// TIA Portal V15.1 export
// export: Created 2024-05-17T05:38:59.7002443Z, ExportSetting WithDefaults, DisplayName Totally Integrated Automation Portal, DisplayVersion V15.1 Update 5, DisplayName TIA Portal Openness, DisplayVersion V15.1 Update 5, DisplayName SINAMICS Startdrive Advanced, DisplayVersion V15.1, DisplayName G130, G150, S120, S150, SINAMICS MV, S210, DisplayVersion V15.1, DisplayName G110M, G120, G120C, G120D, G120P, DisplayVersion V15.1, DisplayName STEP 7 Professional, DisplayVersion V15.1 Update 5, DisplayName STEP 7 Safety, DisplayVersion V15.1, DisplayName WinCC Professional, DisplayVersion V15.1 Update 5, DisplayName SIMATIC Visualization Architect, DisplayVersion V15.1
FUNCTION "209000NCP01ComVD" : Void   // FC256, FBD
TITLE = 209000NCP01ComSafety
{ S7_Optimized_Access := 'FALSE' }
AUTHOR : VCC
VERSION : 0.1
// stored: AutoNumber false, IsIECCheckEnabled false, SetENOAutomatically False, UDAEnableTagReadback false
   VAR_OUTPUT
      O_AlarmA : Bool;   // Alarm A
      O_AlarmB : Bool;   // Alarm B
      O_AlarmC : Bool;   // Alarm C
      O_AlarmD : Bool;   // Alarm D
      O_AlarmABCondition : Bool;   // Alarm AB Condition
      H_IAnim : Word;   // Icon Animation
   END_VAR
BEGIN

REGION Network 1: **** 1 - Inputs **** VD Config Alarm Reporting
   // Communication With VD Alarm Instance
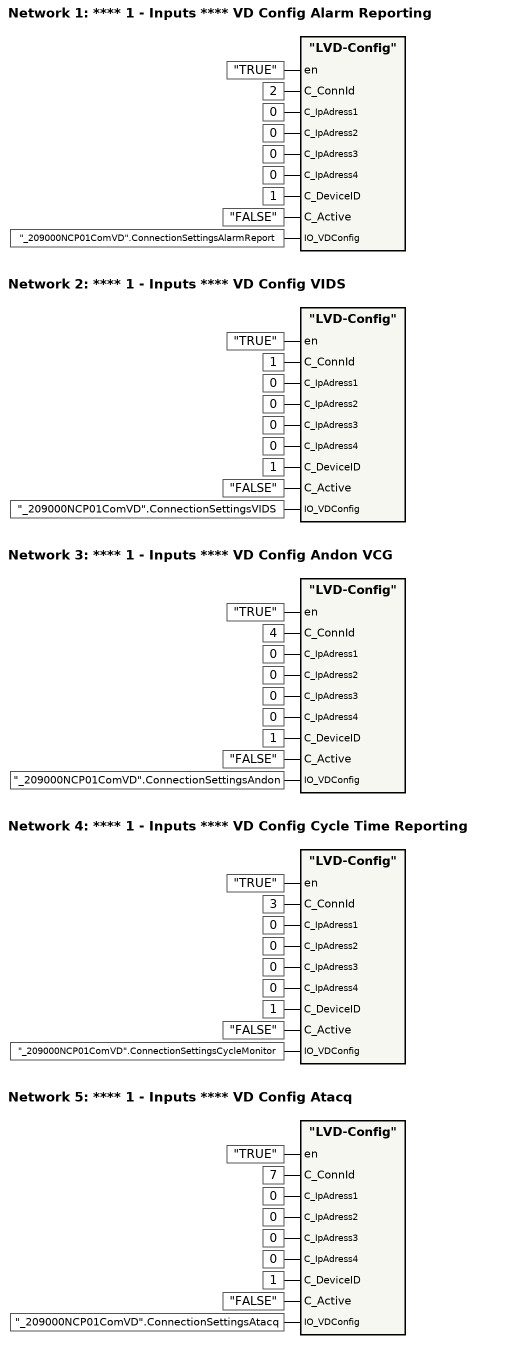
   IF "TRUE" THEN
       "LVD-Config"(C_ConnId := 2,
                    C_IpAdress1 := 0,
                    C_IpAdress2 := 0,
                    C_IpAdress3 := 0,
                    C_IpAdress4 := 0,
                    C_DeviceID := 1,
                    C_Active := "FALSE",
                    IO_VDConfig := "_209000NCP01ComVD".ConnectionSettingsAlarmReport);
   END_IF;
END_REGION

REGION Network 2: **** 1 - Inputs **** VD Config VIDS
   // Communication with VD Prod Instance
   IF "TRUE" THEN
       "LVD-Config"(C_ConnId := 1,
                    C_IpAdress1 := 0,
                    C_IpAdress2 := 0,
                    C_IpAdress3 := 0,
                    C_IpAdress4 := 0,
                    C_DeviceID := 1,
                    C_Active := "FALSE",
                    IO_VDConfig := "_209000NCP01ComVD".ConnectionSettingsVIDS);
   END_IF;
END_REGION

REGION Network 3: **** 1 - Inputs **** VD Config Andon VCG
   // Communication with VD Andon Instance
   IF "TRUE" THEN
       "LVD-Config"(C_ConnId := 4,
                    C_IpAdress1 := 0,
                    C_IpAdress2 := 0,
                    C_IpAdress3 := 0,
                    C_IpAdress4 := 0,
                    C_DeviceID := 1,
                    C_Active := "FALSE",
                    IO_VDConfig := "_209000NCP01ComVD".ConnectionSettingsAndon);
   END_IF;
END_REGION

REGION Network 4: **** 1 - Inputs **** VD Config Cycle Time Reporting
   // Communication setup for cycle time reporting
   IF "TRUE" THEN
       "LVD-Config"(C_ConnId := 3,
                    C_IpAdress1 := 0,
                    C_IpAdress2 := 0,
                    C_IpAdress3 := 0,
                    C_IpAdress4 := 0,
                    C_DeviceID := 1,
                    C_Active := "FALSE",
                    IO_VDConfig := "_209000NCP01ComVD".ConnectionSettingsCycleMonitor);
   END_IF;
END_REGION

REGION Network 5: **** 1 - Inputs **** VD Config Atacq
   // Communication setup for Atacq reporting
   IF "TRUE" THEN
       "LVD-Config"(C_ConnId := 7,
                    C_IpAdress1 := 0,
                    C_IpAdress2 := 0,
                    C_IpAdress3 := 0,
                    C_IpAdress4 := 0,
                    C_DeviceID := 1,
                    C_Active := "FALSE",
                    IO_VDConfig := "_209000NCP01ComVD".ConnectionSettingsAtacq);
   END_IF;
END_REGION

REGION Network 6: **** 1 - Inputs **** VD Config Logistic
   // Communication setup for Logistic reporting
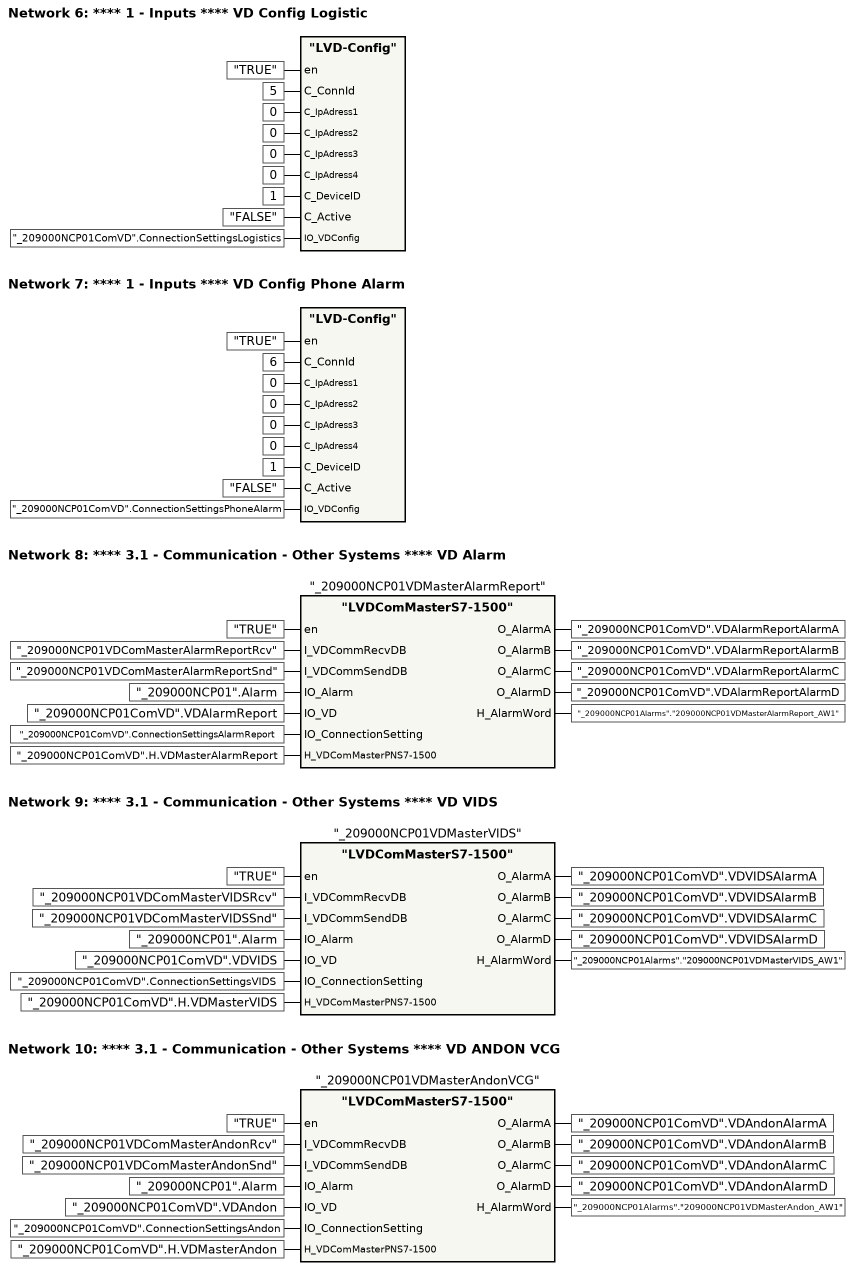
   IF "TRUE" THEN
       "LVD-Config"(C_ConnId := 5,
                    C_IpAdress1 := 0,
                    C_IpAdress2 := 0,
                    C_IpAdress3 := 0,
                    C_IpAdress4 := 0,
                    C_DeviceID := 1,
                    C_Active := "FALSE",
                    IO_VDConfig := "_209000NCP01ComVD".ConnectionSettingsLogistics);
   END_IF;
END_REGION

REGION Network 7: **** 1 - Inputs **** VD Config Phone Alarm
   // Communication setup for Phone Alarm
   IF "TRUE" THEN
       "LVD-Config"(C_ConnId := 6,
                    C_IpAdress1 := 0,
                    C_IpAdress2 := 0,
                    C_IpAdress3 := 0,
                    C_IpAdress4 := 0,
                    C_DeviceID := 1,
                    C_Active := "FALSE",
                    IO_VDConfig := "_209000NCP01ComVD".ConnectionSettingsPhoneAlarm);
   END_IF;
END_REGION

REGION Network 8: **** 3.1 - Communication - Other Systems **** VD Alarm
   // Connection VD Alarm
   IF "TRUE" THEN
       "_209000NCP01VDMasterAlarmReport"(I_VDCommRecvDB := "_209000NCP01VDComMasterAlarmReportRcv",   // "LVDComMasterS7-1500"
                               I_VDCommSendDB := "_209000NCP01VDComMasterAlarmReportSnd",
                               IO_Alarm := "_209000NCP01".Alarm,
                               IO_VD := "_209000NCP01ComVD".VDAlarmReport,
                               IO_ConnectionSetting := "_209000NCP01ComVD".ConnectionSettingsAlarmReport,
                               "H_VDComMasterPNS7-1500" := "_209000NCP01ComVD".H.VDMasterAlarmReport,
                               O_AlarmA => "_209000NCP01ComVD".VDAlarmReportAlarmA,
                               O_AlarmB => "_209000NCP01ComVD".VDAlarmReportAlarmB,
                               O_AlarmC => "_209000NCP01ComVD".VDAlarmReportAlarmC,
                               O_AlarmD => "_209000NCP01ComVD".VDAlarmReportAlarmD,
                               H_AlarmWord => "_209000NCP01Alarms"."209000NCP01VDMasterAlarmReport_AW1");
   END_IF;
END_REGION

REGION Network 9: **** 3.1 - Communication - Other Systems **** VD VIDS
   // Connection VD Production System
   IF "TRUE" THEN
       "_209000NCP01VDMasterVIDS"(I_VDCommRecvDB := "_209000NCP01VDComMasterVIDSRcv",   // "LVDComMasterS7-1500"
                               I_VDCommSendDB := "_209000NCP01VDComMasterVIDSSnd",
                               IO_Alarm := "_209000NCP01".Alarm,
                               IO_VD := "_209000NCP01ComVD".VDVIDS,
                               IO_ConnectionSetting := "_209000NCP01ComVD".ConnectionSettingsVIDS,
                               "H_VDComMasterPNS7-1500" := "_209000NCP01ComVD".H.VDMasterVIDS,
                               O_AlarmA => "_209000NCP01ComVD".VDVIDSAlarmA,
                               O_AlarmB => "_209000NCP01ComVD".VDVIDSAlarmB,
                               O_AlarmC => "_209000NCP01ComVD".VDVIDSAlarmC,
                               O_AlarmD => "_209000NCP01ComVD".VDVIDSAlarmD,
                               H_AlarmWord => "_209000NCP01Alarms"."209000NCP01VDMasterVIDS_AW1");
   END_IF;
END_REGION

REGION Network 10: **** 3.1 - Communication - Other Systems **** VD ANDON VCG
   // Connection VD Andon System
   IF "TRUE" THEN
       "_209000NCP01VDMasterAndonVCG"(I_VDCommRecvDB := "_209000NCP01VDComMasterAndonRcv",   // "LVDComMasterS7-1500"
                               I_VDCommSendDB := "_209000NCP01VDComMasterAndonSnd",
                               IO_Alarm := "_209000NCP01".Alarm,
                               IO_VD := "_209000NCP01ComVD".VDAndon,
                               IO_ConnectionSetting := "_209000NCP01ComVD".ConnectionSettingsAndon,
                               "H_VDComMasterPNS7-1500" := "_209000NCP01ComVD".H.VDMasterAndon,
                               O_AlarmA => "_209000NCP01ComVD".VDAndonAlarmA,
                               O_AlarmB => "_209000NCP01ComVD".VDAndonAlarmB,
                               O_AlarmC => "_209000NCP01ComVD".VDAndonAlarmC,
                               O_AlarmD => "_209000NCP01ComVD".VDAndonAlarmD,
                               H_AlarmWord => "_209000NCP01Alarms"."209000NCP01VDMasterAndon_AW1");
   END_IF;
END_REGION

REGION Network 11: **** 3.1 - Communication - Other Systems **** VD Cycle Time Monitoring
   // Connection VD Cycle Time Monitoring
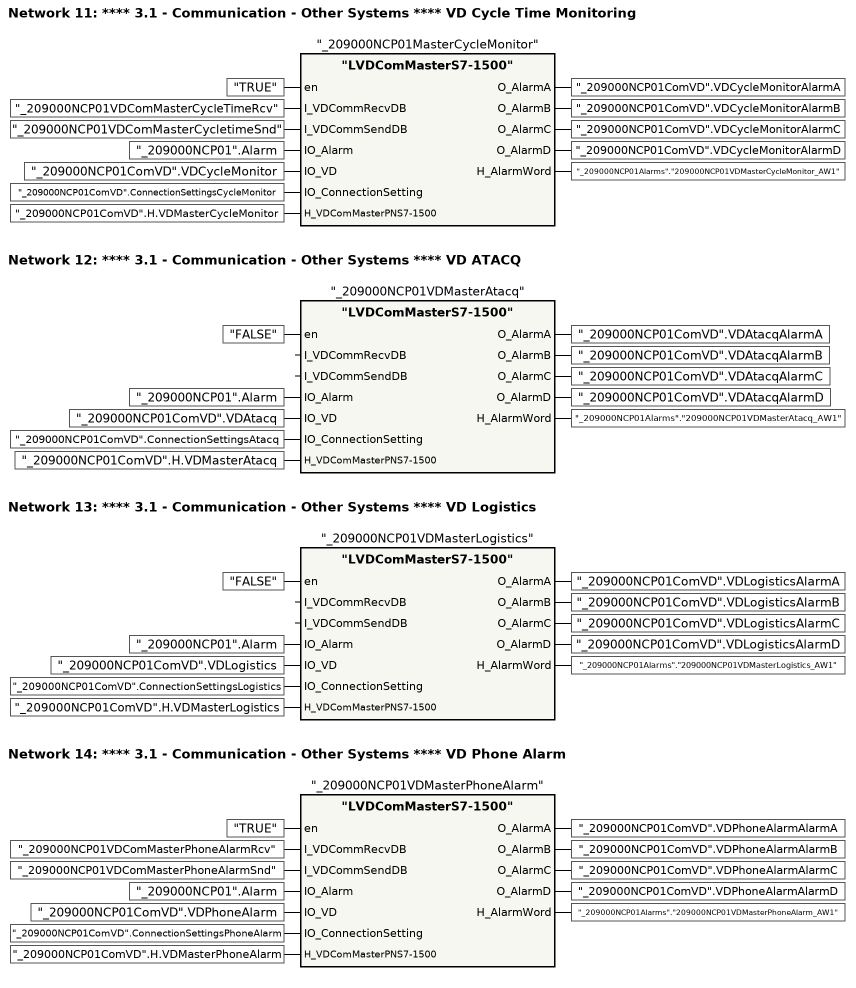
   IF "TRUE" THEN
       "_209000NCP01MasterCycleMonitor"(I_VDCommRecvDB := "_209000NCP01VDComMasterCycleTimeRcv",   // "LVDComMasterS7-1500"
                               I_VDCommSendDB := "_209000NCP01VDComMasterCycletimeSnd",
                               IO_Alarm := "_209000NCP01".Alarm,
                               IO_VD := "_209000NCP01ComVD".VDCycleMonitor,
                               IO_ConnectionSetting := "_209000NCP01ComVD".ConnectionSettingsCycleMonitor,
                               "H_VDComMasterPNS7-1500" := "_209000NCP01ComVD".H.VDMasterCycleMonitor,
                               O_AlarmA => "_209000NCP01ComVD".VDCycleMonitorAlarmA,
                               O_AlarmB => "_209000NCP01ComVD".VDCycleMonitorAlarmB,
                               O_AlarmC => "_209000NCP01ComVD".VDCycleMonitorAlarmC,
                               O_AlarmD => "_209000NCP01ComVD".VDCycleMonitorAlarmD,
                               H_AlarmWord => "_209000NCP01Alarms"."209000NCP01VDMasterCycleMonitor_AW1");
   END_IF;
END_REGION

REGION Network 12: **** 3.1 - Communication - Other Systems **** VD ATACQ
   // Connection VD ATACQ
   IF "FALSE" THEN
       "_209000NCP01VDMasterAtacq"(IO_Alarm := "_209000NCP01".Alarm,   // "LVDComMasterS7-1500"
                               IO_VD := "_209000NCP01ComVD".VDAtacq,
                               IO_ConnectionSetting := "_209000NCP01ComVD".ConnectionSettingsAtacq,
                               "H_VDComMasterPNS7-1500" := "_209000NCP01ComVD".H.VDMasterAtacq,
                               O_AlarmA => "_209000NCP01ComVD".VDAtacqAlarmA,
                               O_AlarmB => "_209000NCP01ComVD".VDAtacqAlarmB,
                               O_AlarmC => "_209000NCP01ComVD".VDAtacqAlarmC,
                               O_AlarmD => "_209000NCP01ComVD".VDAtacqAlarmD,
                               H_AlarmWord => "_209000NCP01Alarms"."209000NCP01VDMasterAtacq_AW1");
   END_IF;
END_REGION

REGION Network 13: **** 3.1 - Communication - Other Systems **** VD Logistics
   // Connection VD Logistics
   IF "FALSE" THEN
       "_209000NCP01VDMasterLogistics"(IO_Alarm := "_209000NCP01".Alarm,   // "LVDComMasterS7-1500"
                               IO_VD := "_209000NCP01ComVD".VDLogistics,
                               IO_ConnectionSetting := "_209000NCP01ComVD".ConnectionSettingsLogistics,
                               "H_VDComMasterPNS7-1500" := "_209000NCP01ComVD".H.VDMasterLogistics,
                               O_AlarmA => "_209000NCP01ComVD".VDLogisticsAlarmA,
                               O_AlarmB => "_209000NCP01ComVD".VDLogisticsAlarmB,
                               O_AlarmC => "_209000NCP01ComVD".VDLogisticsAlarmC,
                               O_AlarmD => "_209000NCP01ComVD".VDLogisticsAlarmD,
                               H_AlarmWord => "_209000NCP01Alarms"."209000NCP01VDMasterLogistics_AW1");
   END_IF;
END_REGION

REGION Network 14: **** 3.1 - Communication - Other Systems **** VD Phone Alarm
   // Connection VD Phone Alarm
   IF "TRUE" THEN
       "_209000NCP01VDMasterPhoneAlarm"(I_VDCommRecvDB := "_209000NCP01VDComMasterPhoneAlarmRcv",   // "LVDComMasterS7-1500"
                               I_VDCommSendDB := "_209000NCP01VDComMasterPhoneAlarmSnd",
                               IO_Alarm := "_209000NCP01".Alarm,
                               IO_VD := "_209000NCP01ComVD".VDPhoneAlarm,
                               IO_ConnectionSetting := "_209000NCP01ComVD".ConnectionSettingsPhoneAlarm,
                               "H_VDComMasterPNS7-1500" := "_209000NCP01ComVD".H.VDMasterPhoneAlarm,
                               O_AlarmA => "_209000NCP01ComVD".VDPhoneAlarmAlarmA,
                               O_AlarmB => "_209000NCP01ComVD".VDPhoneAlarmAlarmB,
                               O_AlarmC => "_209000NCP01ComVD".VDPhoneAlarmAlarmC,
                               O_AlarmD => "_209000NCP01ComVD".VDPhoneAlarmAlarmD,
                               H_AlarmWord => "_209000NCP01Alarms"."209000NCP01VDMasterPhoneAlarm_AW1");
   END_IF;
END_REGION

REGION Network 15: **** 3.1 - Communication - Other Systems **** Phone Alarm Request
   // Phone alarm request
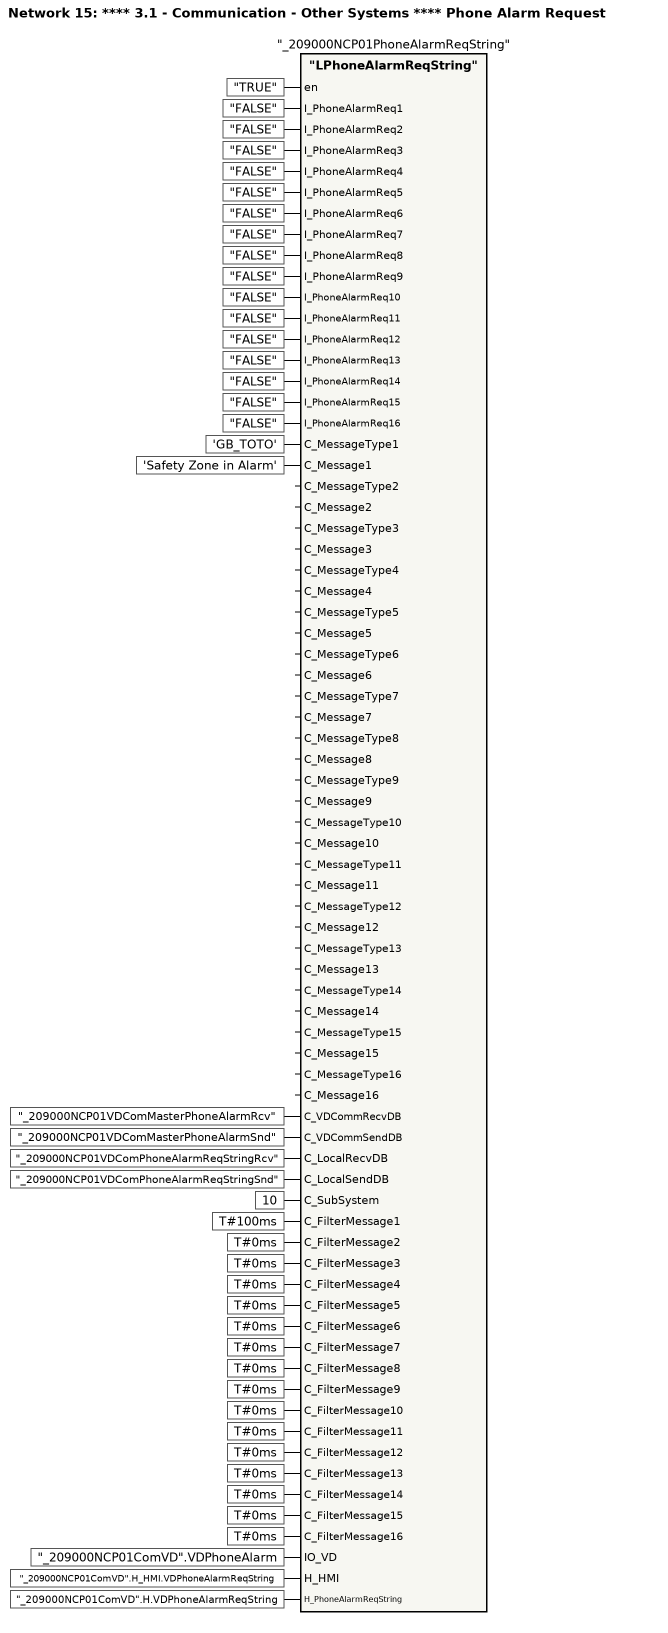
   IF "TRUE" THEN
       "_209000NCP01PhoneAlarmReqString"(I_PhoneAlarmReq1 := "FALSE",   // "LPhoneAlarmReqString"
                               I_PhoneAlarmReq2 := "FALSE",
                               I_PhoneAlarmReq3 := "FALSE",
                               I_PhoneAlarmReq4 := "FALSE",
                               I_PhoneAlarmReq5 := "FALSE",
                               I_PhoneAlarmReq6 := "FALSE",
                               I_PhoneAlarmReq7 := "FALSE",
                               I_PhoneAlarmReq8 := "FALSE",
                               I_PhoneAlarmReq9 := "FALSE",
                               I_PhoneAlarmReq10 := "FALSE",
                               I_PhoneAlarmReq11 := "FALSE",
                               I_PhoneAlarmReq12 := "FALSE",
                               I_PhoneAlarmReq13 := "FALSE",
                               I_PhoneAlarmReq14 := "FALSE",
                               I_PhoneAlarmReq15 := "FALSE",
                               I_PhoneAlarmReq16 := "FALSE",
                               C_MessageType1 := 'GB_TOTO',
                               C_Message1 := 'Safety Zone in Alarm',
                               C_VDCommRecvDB := "_209000NCP01VDComMasterPhoneAlarmRcv",
                               C_VDCommSendDB := "_209000NCP01VDComMasterPhoneAlarmSnd",
                               C_LocalRecvDB := "_209000NCP01VDComPhoneAlarmReqStringRcv",
                               C_LocalSendDB := "_209000NCP01VDComPhoneAlarmReqStringSnd",
                               C_SubSystem := 10,
                               C_FilterMessage1 := T#100ms,
                               C_FilterMessage2 := T#0ms,
                               C_FilterMessage3 := T#0ms,
                               C_FilterMessage4 := T#0ms,
                               C_FilterMessage5 := T#0ms,
                               C_FilterMessage6 := T#0ms,
                               C_FilterMessage7 := T#0ms,
                               C_FilterMessage8 := T#0ms,
                               C_FilterMessage9 := T#0ms,
                               C_FilterMessage10 := T#0ms,
                               C_FilterMessage11 := T#0ms,
                               C_FilterMessage12 := T#0ms,
                               C_FilterMessage13 := T#0ms,
                               C_FilterMessage14 := T#0ms,
                               C_FilterMessage15 := T#0ms,
                               C_FilterMessage16 := T#0ms,
                               IO_VD := "_209000NCP01ComVD".VDPhoneAlarm,
                               H_HMI := "_209000NCP01ComVD".H_HMI.VDPhoneAlarmReqString,
                               H_PhoneAlarmReqString := "_209000NCP01ComVD".H.VDPhoneAlarmReqString);
   END_IF;
END_REGION

REGION Network 16: **** 4.6 - Machine status - Indications **** Icon animation
   // Icon animation to WinCC
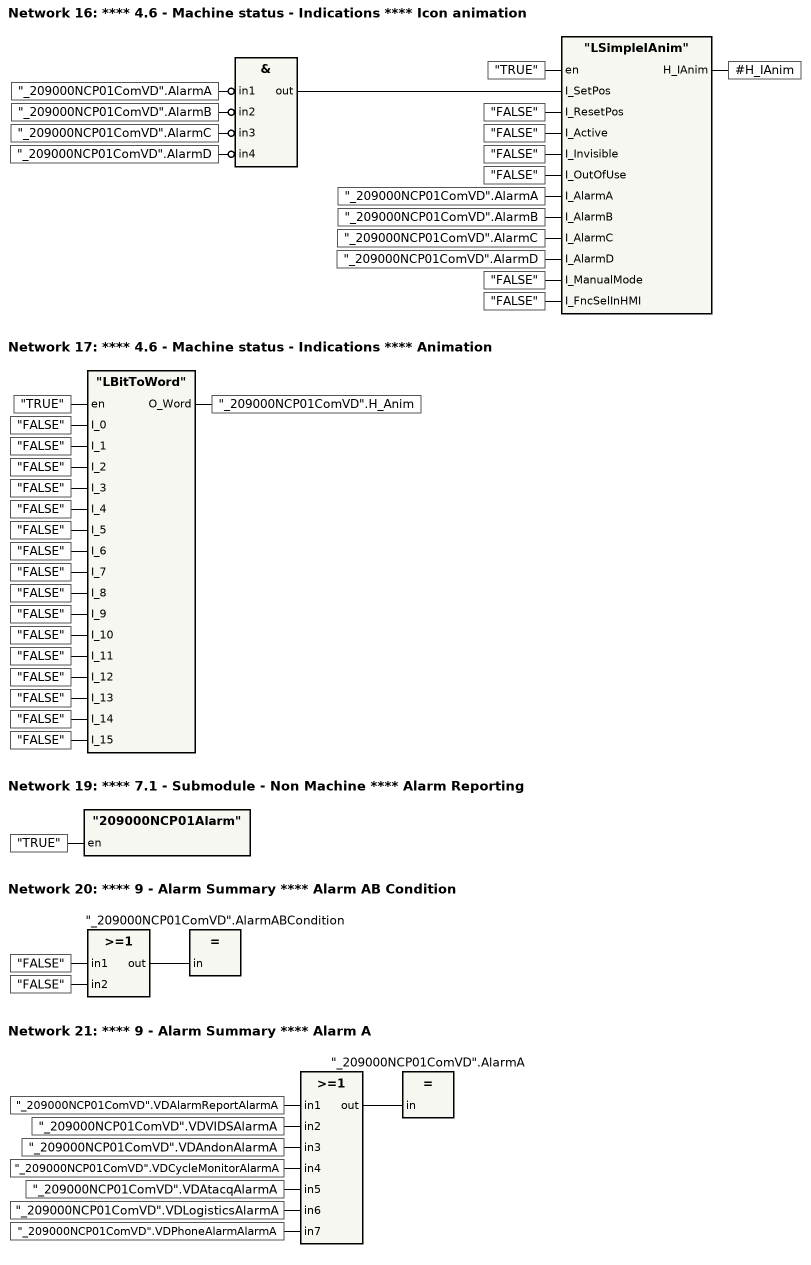
   IF "TRUE" THEN
       "LSimpleIAnim"(I_SetPos := NOT "_209000NCP01ComVD".AlarmA AND NOT "_209000NCP01ComVD".AlarmB AND NOT "_209000NCP01ComVD".AlarmC AND NOT "_209000NCP01ComVD".AlarmD,
                      I_ResetPos := "FALSE",
                      I_Active := "FALSE",
                      I_Invisible := "FALSE",
                      I_OutOfUse := "FALSE",
                      I_AlarmA := "_209000NCP01ComVD".AlarmA,
                      I_AlarmB := "_209000NCP01ComVD".AlarmB,
                      I_AlarmC := "_209000NCP01ComVD".AlarmC,
                      I_AlarmD := "_209000NCP01ComVD".AlarmD,
                      I_ManualMode := "FALSE",
                      I_FncSelInHMI := "FALSE",
                      H_IAnim => #H_IAnim);
   END_IF;
END_REGION

REGION Network 17: **** 4.6 - Machine status - Indications **** Animation
   // Animation
   IF "TRUE" THEN
       "LBitToWord"(I_0 := "FALSE",
                    I_1 := "FALSE",
                    I_2 := "FALSE",
                    I_3 := "FALSE",
                    I_4 := "FALSE",
                    I_5 := "FALSE",
                    I_6 := "FALSE",
                    I_7 := "FALSE",
                    I_8 := "FALSE",
                    I_9 := "FALSE",
                    I_10 := "FALSE",
                    I_11 := "FALSE",
                    I_12 := "FALSE",
                    I_13 := "FALSE",
                    I_14 := "FALSE",
                    I_15 := "FALSE",
                    O_Word => "_209000NCP01ComVD".H_Anim);
   END_IF;
END_REGION

NETWORK
TITLE = **** 4.6 - Machine Status - Indications **** Animation DB number
// DB number
      OPN   "_209000NCP01ComVD";
      L     DBNO;
      T     "_209000NCP01ComVD".H_DBnr;

REGION Network 19: **** 7.1 - Submodule - Non Machine **** Alarm Reporting
   // Alarm Handler MES System
   IF "TRUE" THEN "209000NCP01Alarm"(); END_IF;
END_REGION

REGION Network 20: **** 9 - Alarm Summary **** Alarm AB Condition
   // Alarm AB Condition
   "_209000NCP01ComVD".AlarmABCondition := "FALSE" OR "FALSE";
END_REGION

REGION Network 21: **** 9 - Alarm Summary **** Alarm A
   // Summary of Alarm A
   "_209000NCP01ComVD".AlarmA := "_209000NCP01ComVD".VDAlarmReportAlarmA OR "_209000NCP01ComVD".VDVIDSAlarmA OR "_209000NCP01ComVD".VDAndonAlarmA OR "_209000NCP01ComVD".VDCycleMonitorAlarmA OR "_209000NCP01ComVD".VDAtacqAlarmA OR "_209000NCP01ComVD".VDLogisticsAlarmA OR "_209000NCP01ComVD".VDPhoneAlarmAlarmA;
END_REGION

REGION Network 22: **** 9 - Alarm Summary **** Alarm B
   // Summary of Alarm B
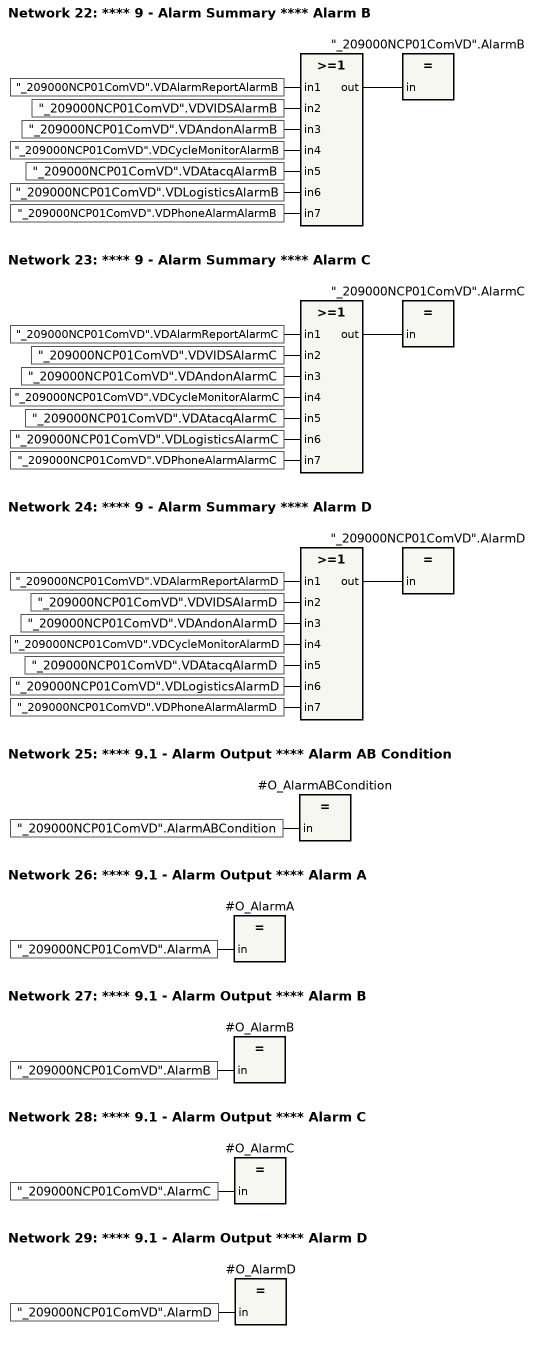
   "_209000NCP01ComVD".AlarmB := "_209000NCP01ComVD".VDAlarmReportAlarmB OR "_209000NCP01ComVD".VDVIDSAlarmB OR "_209000NCP01ComVD".VDAndonAlarmB OR "_209000NCP01ComVD".VDCycleMonitorAlarmB OR "_209000NCP01ComVD".VDAtacqAlarmB OR "_209000NCP01ComVD".VDLogisticsAlarmB OR "_209000NCP01ComVD".VDPhoneAlarmAlarmB;
END_REGION

REGION Network 23: **** 9 - Alarm Summary **** Alarm C
   // Summary of Alarm C
   "_209000NCP01ComVD".AlarmC := "_209000NCP01ComVD".VDAlarmReportAlarmC OR "_209000NCP01ComVD".VDVIDSAlarmC OR "_209000NCP01ComVD".VDAndonAlarmC OR "_209000NCP01ComVD".VDCycleMonitorAlarmC OR "_209000NCP01ComVD".VDAtacqAlarmC OR "_209000NCP01ComVD".VDLogisticsAlarmC OR "_209000NCP01ComVD".VDPhoneAlarmAlarmC;
END_REGION

REGION Network 24: **** 9 - Alarm Summary **** Alarm D
   // Summary of Alarm D
   "_209000NCP01ComVD".AlarmD := "_209000NCP01ComVD".VDAlarmReportAlarmD OR "_209000NCP01ComVD".VDVIDSAlarmD OR "_209000NCP01ComVD".VDAndonAlarmD OR "_209000NCP01ComVD".VDCycleMonitorAlarmD OR "_209000NCP01ComVD".VDAtacqAlarmD OR "_209000NCP01ComVD".VDLogisticsAlarmD OR "_209000NCP01ComVD".VDPhoneAlarmAlarmD;
END_REGION

REGION Network 25: **** 9.1 - Alarm Output **** Alarm AB Condition
   // Alarm AB ConditionAlarm A
   #O_AlarmABCondition := "_209000NCP01ComVD".AlarmABCondition;
END_REGION

REGION Network 26: **** 9.1 - Alarm Output **** Alarm A
   // Alarm A
   #O_AlarmA := "_209000NCP01ComVD".AlarmA;
END_REGION

REGION Network 27: **** 9.1 - Alarm Output **** Alarm B
   // Alarm B
   #O_AlarmB := "_209000NCP01ComVD".AlarmB;
END_REGION

REGION Network 28: **** 9.1 - Alarm Output **** Alarm C
   // Alarm C
   #O_AlarmC := "_209000NCP01ComVD".AlarmC;
END_REGION

REGION Network 29: **** 9.1 - Alarm Output **** Alarm D
   // Alarm D
   #O_AlarmD := "_209000NCP01ComVD".AlarmD;
END_REGION

REGION Network 30: **** 9.2 - Alarm DWord**** Alarm To DWord
   // Alarm Word
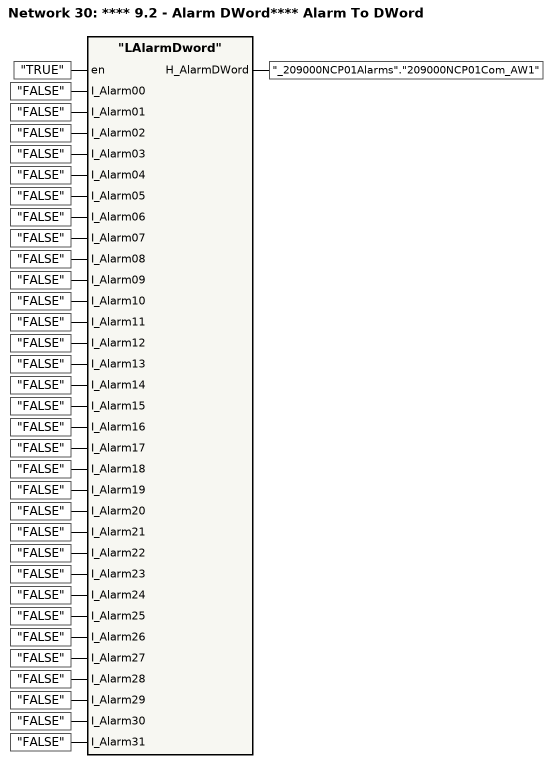
   IF "TRUE" THEN
       "LAlarmDword"(I_Alarm00 := "FALSE",
                     I_Alarm01 := "FALSE",
                     I_Alarm02 := "FALSE",
                     I_Alarm03 := "FALSE",
                     I_Alarm04 := "FALSE",
                     I_Alarm05 := "FALSE",
                     I_Alarm06 := "FALSE",
                     I_Alarm07 := "FALSE",
                     I_Alarm08 := "FALSE",
                     I_Alarm09 := "FALSE",
                     I_Alarm10 := "FALSE",
                     I_Alarm11 := "FALSE",
                     I_Alarm12 := "FALSE",
                     I_Alarm13 := "FALSE",
                     I_Alarm14 := "FALSE",
                     I_Alarm15 := "FALSE",
                     I_Alarm16 := "FALSE",
                     I_Alarm17 := "FALSE",
                     I_Alarm18 := "FALSE",
                     I_Alarm19 := "FALSE",
                     I_Alarm20 := "FALSE",
                     I_Alarm21 := "FALSE",
                     I_Alarm22 := "FALSE",
                     I_Alarm23 := "FALSE",
                     I_Alarm24 := "FALSE",
                     I_Alarm25 := "FALSE",
                     I_Alarm26 := "FALSE",
                     I_Alarm27 := "FALSE",
                     I_Alarm28 := "FALSE",
                     I_Alarm29 := "FALSE",
                     I_Alarm30 := "FALSE",
                     I_Alarm31 := "FALSE",
                     H_AlarmDWord => "_209000NCP01Alarms"."209000NCP01Com_AW1");
   END_IF;
END_REGION
END_FUNCTION
